# EPICS autosave request: linkamT96App/Db/LinkamRHGen_settings.req
$(P):STARTHUM.VAL
$(P):HUMIDITY:SET.VAL
$(P):HUMIDITY.SCAN
$(P):HUMIDITY:TEMP.SCAN
